% RSLogix 500 project Project_10.RSS, saved by version 8.30.00.16 %
PROJECT "UNTITLED"    % processor: Bul.1763 MicroLogix 1100 Series B %

PROGRAM FILES
  LAD 2   3 rungs
  LAD 3 "IO"  7 rungs  % Input/Output %
  LAD 4 "LOGIC"  17 rungs

DATA FILES
  O0 OUTPUT  4 elements
  I1 INPUT  6 elements
  S2 STATUS  66 elements
  B3 BINARY  3 elements
  T4 TIMER  4 elements
  C5 COUNTER  1 elements
  R6 CONTROL  1 elements
  N7 INTEGER  20 elements
  F8 FLOAT  1 elements

LADDER 2
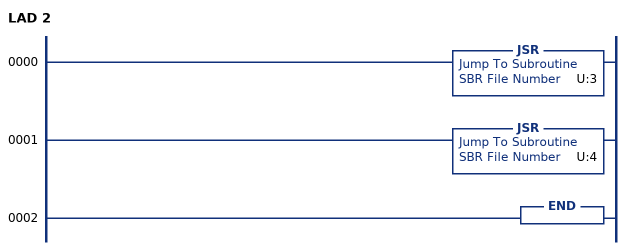
% Rung: 0 %
SOR JSR U:3 EOR
% Rung: 1 %
SOR JSR U:4 EOR
% Rung: 2 %
SOR END EOR

LADDER 3 "IO"    % Input/Output %
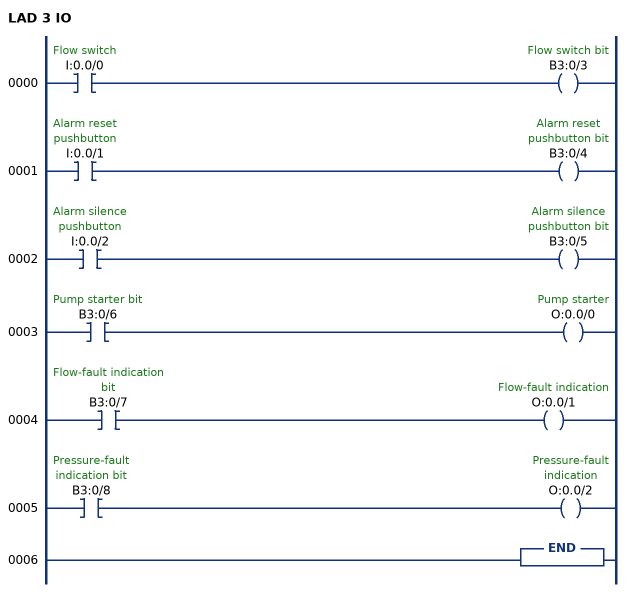
% Rung: 0 %
SOR XIC I:0.0/0 OTE B3:0/3 EOR
%   I:0.0/0  "Flow switch" %
%   B3:0/3  "Flow switch bit" %
% Rung: 1 %
SOR XIC I:0.0/1 OTE B3:0/4 EOR
%   I:0.0/1  "Alarm reset pushbutton" %
%   B3:0/4  "Alarm reset pushbutton bit" %
% Rung: 2 %
SOR XIC I:0.0/2 OTE B3:0/5 EOR
%   I:0.0/2  "Alarm silence pushbutton" %
%   B3:0/5  "Alarm silence pushbutton bit" %
% Rung: 3 %
SOR XIC B3:0/6 OTE O:0.0/0 EOR
%   B3:0/6  "Pump starter bit" %
%   O:0.0/0  "Pump starter" %
% Rung: 4 %
SOR XIC B3:0/7 OTE O:0.0/1 EOR
%   B3:0/7  "Flow-fault indication bit" %
%   O:0.0/1  "Flow-fault indication" %
% Rung: 5 %
SOR XIC B3:0/8 OTE O:0.0/2 EOR
%   B3:0/8  "Pressure-fault indication bit" %
%   O:0.0/2  "Pressure-fault indication" %
% Rung: 6 %
SOR END EOR

LADDER 4 "LOGIC"
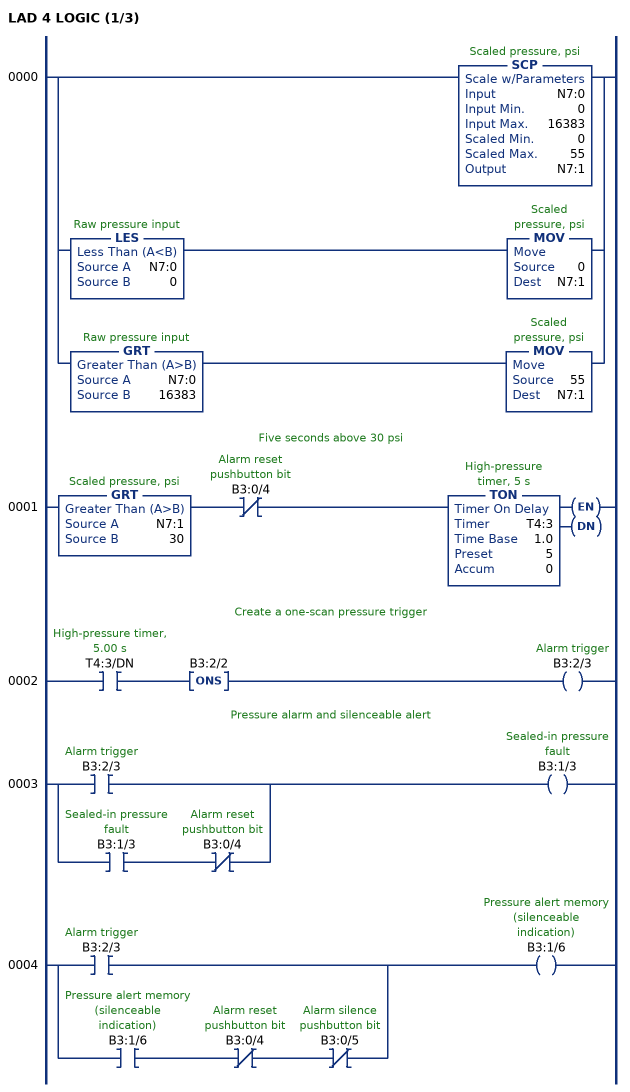
% Rung: 0 %
SOR BST SCP N7:0 0 16383 0 55 N7:1 NXB LES N7:0 0 MOV 0 N7:1 NXB GRT N7:0 16383 MOV 55 N7:1 BND EOR
%   N7:0  "Raw pressure input" %
%   N7:1  "Scaled pressure, psi" %
% Rung: 1 %
% Five seconds above 30 psi %
SOR GRT N7:1 30 XIO B3:0/4 TON T4:3 1.0 5 0 EOR
%   N7:1  "Scaled pressure, psi" %
%   B3:0/4  "Alarm reset pushbutton bit" %
%   T4:3  "High-pressure timer, 5 s" %
% Rung: 2 %
% Create a one-scan pressure trigger %
SOR XIC T4:3/DN ONS B3:2/2 OTE B3:2/3 EOR
%   T4:3/DN  "High-pressure timer, 5.00 s" %
%   B3:2/3  "Alarm trigger" %
% Rung: 3 %
% Pressure alarm and silenceable alert %
SOR BST XIC B3:2/3 NXB XIC B3:1/3 XIO B3:0/4 BND OTE B3:1/3 EOR
%   B3:2/3  "Alarm trigger" %
%   B3:1/3  "Sealed-in pressure fault" %
%   B3:0/4  "Alarm reset pushbutton bit" %
% Rung: 4 %
SOR BST XIC B3:2/3 NXB XIC B3:1/6 XIO B3:0/4 XIO B3:0/5 BND OTE B3:1/6 EOR
%   B3:2/3  "Alarm trigger" %
%   B3:1/6  "Pressure alert memory (silenceable indication)" %
%   B3:0/4  "Alarm reset pushbutton bit" %
%   B3:0/5  "Alarm silence pushbutton bit" %

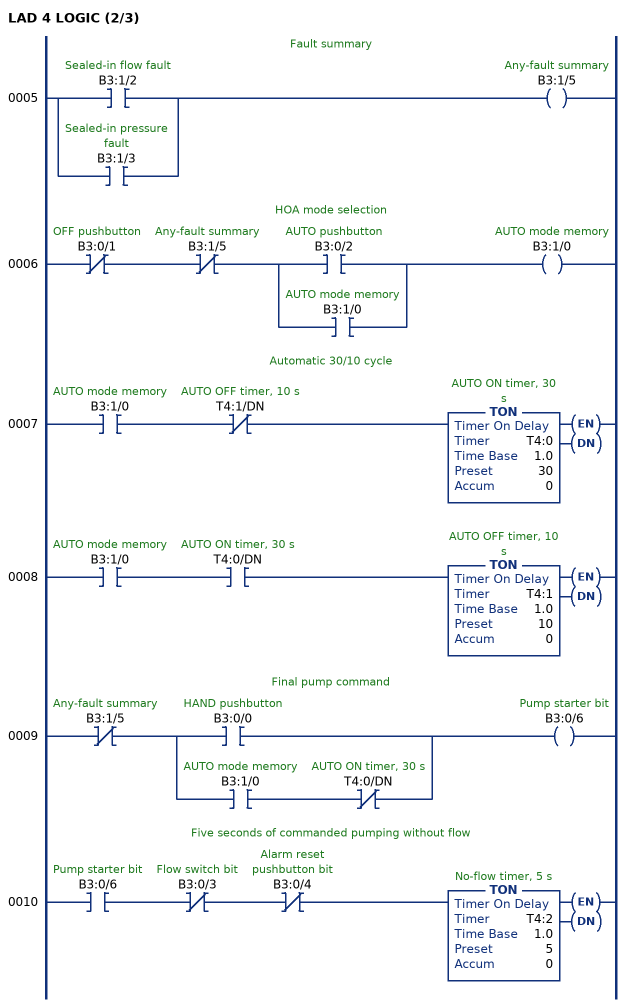
% Rung: 5 %
% Fault summary %
SOR BST XIC B3:1/2 NXB XIC B3:1/3 BND OTE B3:1/5 EOR
%   B3:1/2  "Sealed-in flow fault" %
%   B3:1/3  "Sealed-in pressure fault" %
%   B3:1/5  "Any-fault summary" %
% Rung: 6 %
% HOA mode selection %
SOR XIO B3:0/1 XIO B3:1/5 BST XIC B3:0/2 NXB XIC B3:1/0 BND OTE B3:1/0 EOR
%   B3:0/1  "OFF pushbutton" %
%   B3:1/5  "Any-fault summary" %
%   B3:0/2  "AUTO pushbutton" %
%   B3:1/0  "AUTO mode memory" %
% Rung: 7 %
% Automatic 30/10 cycle %
SOR XIC B3:1/0 XIO T4:1/DN TON T4:0 1.0 30 0 EOR
%   B3:1/0  "AUTO mode memory" %
%   T4:1  "AUTO OFF timer, 10 s" %
%   T4:0  "AUTO ON timer, 30 s" %
% Rung: 8 %
SOR XIC B3:1/0 XIC T4:0/DN TON T4:1 1.0 10 0 EOR
%   B3:1/0  "AUTO mode memory" %
%   T4:0  "AUTO ON timer, 30 s" %
%   T4:1  "AUTO OFF timer, 10 s" %
% Rung: 9 %
% Final pump command %
SOR XIO B3:1/5 BST XIC B3:0/0 NXB XIC B3:1/0 XIO T4:0/DN BND OTE B3:0/6 EOR
%   B3:1/5  "Any-fault summary" %
%   B3:0/0  "HAND pushbutton" %
%   B3:1/0  "AUTO mode memory" %
%   T4:0  "AUTO ON timer, 30 s" %
%   B3:0/6  "Pump starter bit" %
% Rung: 10 %
% Five seconds of commanded pumping without flow %
SOR XIC B3:0/6 XIO B3:0/3 XIO B3:0/4 TON T4:2 1.0 5 0 EOR
%   B3:0/6  "Pump starter bit" %
%   B3:0/3  "Flow switch bit" %
%   B3:0/4  "Alarm reset pushbutton bit" %
%   T4:2  "No-flow timer, 5 s" %

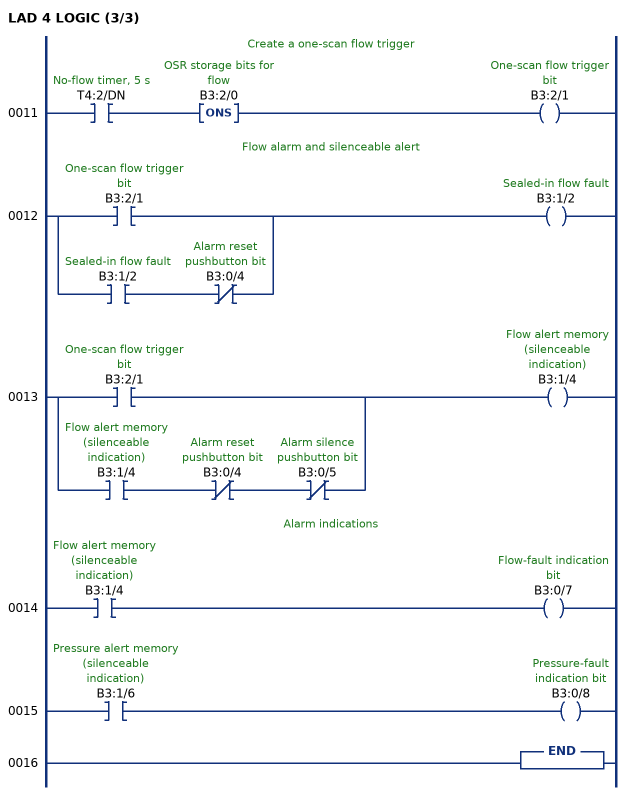
% Rung: 11 %
% Create a one-scan flow trigger %
SOR XIC T4:2/DN ONS B3:2/0 OTE B3:2/1 EOR
%   T4:2  "No-flow timer, 5 s" %
%   B3:2/0  "OSR storage bits for flow" %
%   B3:2/1  "One-scan flow trigger bit" %
% Rung: 12 %
% Flow alarm and silenceable alert %
SOR BST XIC B3:2/1 NXB XIC B3:1/2 XIO B3:0/4 BND OTE B3:1/2 EOR
%   B3:2/1  "One-scan flow trigger bit" %
%   B3:1/2  "Sealed-in flow fault" %
%   B3:0/4  "Alarm reset pushbutton bit" %
% Rung: 13 %
SOR BST XIC B3:2/1 NXB XIC B3:1/4 XIO B3:0/4 XIO B3:0/5 BND OTE B3:1/4 EOR
%   B3:2/1  "One-scan flow trigger bit" %
%   B3:1/4  "Flow alert memory (silenceable indication)" %
%   B3:0/4  "Alarm reset pushbutton bit" %
%   B3:0/5  "Alarm silence pushbutton bit" %
% Rung: 14 %
% Alarm indications %
SOR XIC B3:1/4 OTE B3:0/7 EOR
%   B3:1/4  "Flow alert memory (silenceable indication)" %
%   B3:0/7  "Flow-fault indication bit" %
% Rung: 15 %
SOR XIC B3:1/6 OTE B3:0/8 EOR
%   B3:1/6  "Pressure alert memory (silenceable indication)" %
%   B3:0/8  "Pressure-fault indication bit" %
% Rung: 16 %
SOR END EOR

DATA TABLE (non-zero values as saved)
DATA B3
% B3:0 % 0X000E 0X0000 0X0000
DATA T4
% .PRE .ACC %
% T4:0 % 30 0
% T4:1 % 10 0
% T4:2 % 5 0
% T4:3 % 5 0
DATA N7
% N7:0 % 8000 27 0 0 0 0 0 0 0 0
